(* IEC 61131-3 sources: IEC61131-3-CDSV3/Regular Expressions/src, 1 file *)

(* ---- ParameterList.gvl ---- *)
(*#-#-#-#-#-#-#-#-#-#---Declaration---#-#-#-#-#-#-#-#-#-#-#-#-#*)

{attribute 'qualified_only'}
VAR_GLOBAL CONSTANT
    uiMaxPatternTokens: UINT := 255;    // The maximum amount of tokens to support parsing (compiling) - the counting starts from 0, so add 1 to the number in your mind
END_VAR
